// TIA Portal V16 export
// export: Created 2021-11-12T13:31:14.2602754Z, ExportSetting WithDefaults, DisplayName Totally Integrated Automation Portal, DisplayVersion V16 Update 3, DisplayName TIA Portal Version Control Interface, DisplayVersion V16 Update 2, DisplayName TIA Portal Openness, DisplayVersion V16 Update 3, DisplayName SINAMICS Startdrive Advanced, DisplayVersion V16 Update 5, DisplayName SINAMICS Startdrive G130, G150, S120, S150, SINAMICS MV, S210, DisplayVersion V16 Update 5, DisplayName SINAMICS Startdrive G110M, G120, G120C, G120D, G120P, G115D, DisplayVersion V16 Update 5, DisplayName STEP 7 Professional, DisplayVersion V16 Update 3, DisplayName STEP 7 Safety, DisplayVersion V16, DisplayName WinCC UA Professional, DisplayVersion V16 Update 3
FUNCTION_BLOCK "STD_EuchnerSafetySwitch2MBM"   // FB84, LAD
TITLE = Euchner safety switch 2 Main module / Euchner bezpečnostní zámek 2 hlavní modul
{ S7_Optimized_Access := 'TRUE' }
VERSION : 0.1
// MICE STD Function Block
// STD_EuchnerSafetySwitch2 MBM module
// 
// Version                             Creation date                       Created by
// 0.1                                     16.8.2019                                ZS
// stored: AutoNumber true, IsIECCheckEnabled false, IsRetainMemResEnabled false, MemoryReserve 100, SetENOAutomatically false, UDAEnableTagReadback false
   VAR_INPUT
      IS_ZoneM { ExternalAccessible := 'False'; ExternalVisible := 'False'; ExternalWritable := 'False'} : "UDT_Status_main";   // Main structure from zone / Main struktura ze zóny
      IS_ZoneS { ExternalAccessible := 'False'; ExternalVisible := 'False'; ExternalWritable := 'False'} : "UDT_Zone_Status_specific";   // Specific structure from zone / Specific struktura zóny
      IB1ResetLock : Bool;   // Reset errors and lock / Reset chyby a zamknutí
      IB1AlarmSuppress : Bool;   // Alarm suppression - external / Potlačení poruch
      IB_DoorMBMData : "UDT_MBM_Extended.Input";   // Vstupní data z modulu MBM / Input data from module
   END_VAR
   VAR_OUTPUT
      OS_Status : Struct
         Main : "UDT_Status_main";
         Specific : "UDT_EuchnerSafetySwitch2MBM_Status_Specific";
         Error : "UDT_Error01";
      END_STRUCT;
      OB_DoorMBMReset : Bool;   // Reset output byte for MBM module / Reset výstupního bitu pro MBM modul
   END_VAR
   VAR
      SS_Alarm : Struct   // Device alarms / Zařízení poruchy
         DoorMainModule : Bool;   // Door main module / Dveře hlavní modul
         DoorModule1 : Bool;   // Door module 1 / Dveře modul 1
         DoorModule2 : Bool;   // Dveře modul 2 / Door module 2
         DoorOverallSystem : Bool;   // Dveře nadřazený systém / Door overall system
         Res_0_4 : Bool;
         Res_0_5 : Bool;
         Res_0_6 : Bool;
         Res_0_7 : Bool;
         Res_1_0 : Bool;
         Res_1_1 : Bool;
         Res_1_2 : Bool;
         Res_1_3 : Bool;
         Res_1_4 : Bool;
         Res_1_5 : Bool;
         Res_1_6 : Bool;
         Res_1_7 : Bool;
      END_STRUCT;
      SS_Warning : Struct   // Device warnings / Zařízení varování
         Res_0_0 : Bool;
         Res_0_1 : Bool;
         Res_0_2 : Bool;
         Res_0_3 : Bool;
         Res_0_4 : Bool;
         Res_0_5 : Bool;
         Res_0_6 : Bool;
         Res_0_7 : Bool;
         Res_1_0 : Bool;
         Res_1_1 : Bool;
         Res_1_2 : Bool;
         Res_1_3 : Bool;
         Res_1_4 : Bool;
         Res_1_5 : Bool;
         Res_1_6 : Bool;
         Res_1_7 : Bool;
      END_STRUCT;
      SB1CollError : Bool;   // Collective error from device / Sumace poruchy zařízení
      ST_TONExtensAck { S7_SetPoint := 'True'} : TON_TIME;   // Časovač pro prodloužení pulsu / Timer for extension pulse
      SB_DoorMBMReset : Bool;   // Reset output byte for MBM module / Reset výstupního bitu pro MBM modulu
      SB1Reset : Bool;   // Reset errors and lock / Reset chyby a zamknutí
      SB1ResetEdge : Bool;   // Edge reset errors and lock / Hrana resetu poruchy a zamknutí
   END_VAR
   VAR_TEMP
      TS_Status : Struct
         Main : "UDT_Status_main";
         Specific : "UDT_EuchnerSafetySwitch2MBM_Status_Specific";
         Error : "UDT_Error01";
      END_STRUCT;
      TS_Command : "UDT_EuchnerSafetySwitch2MBM_Command";
      TS_Parameter : "UDT_EuchnerSafetySwitch2MBM_Parameter";
   END_VAR
   VAR_TEMP   // added for the SCL form of the ladder/FBD networks
      _w1 : Bool;
   END_VAR
BEGIN

REGION Network 1: Clear temporary TS_Status - Main, Specific / Mazání dočasných TS_Status - Main, Specific
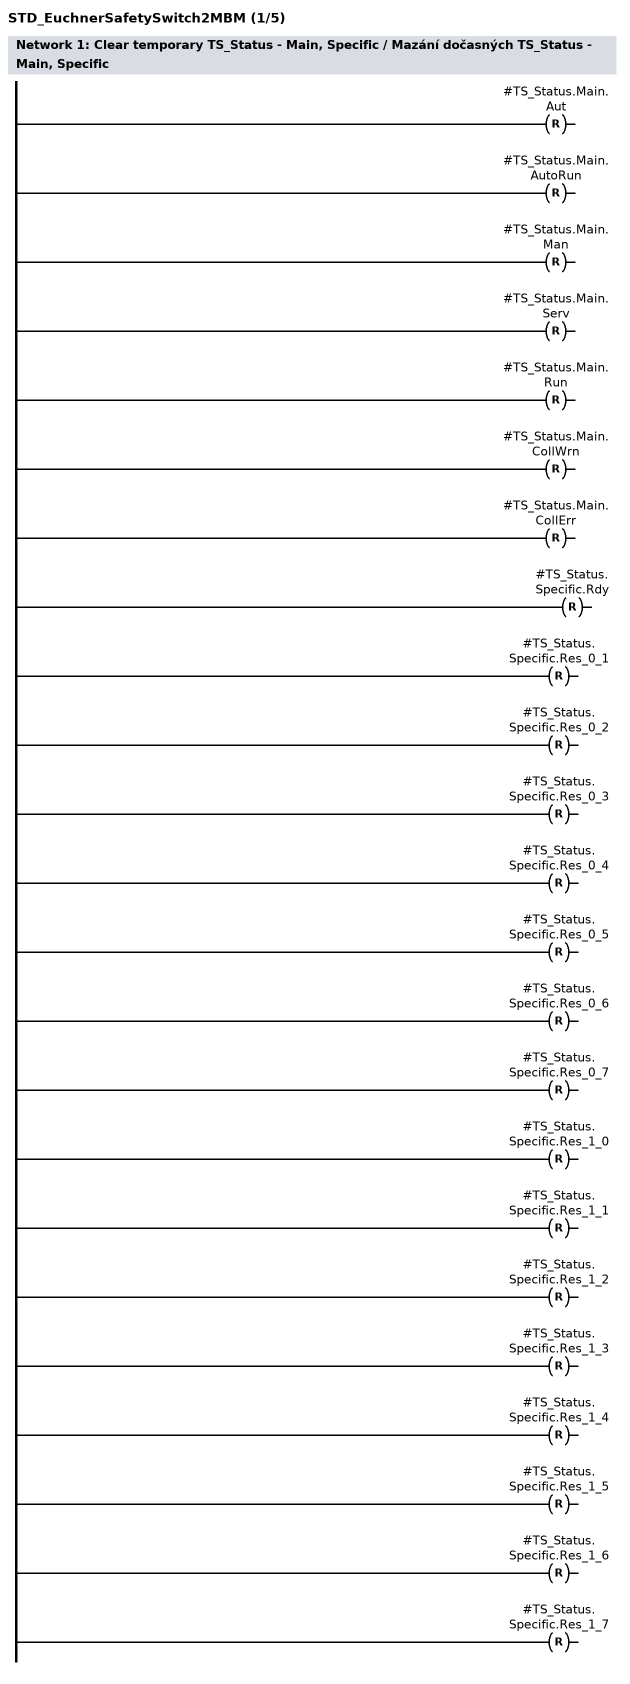
   RUNG wire#powerrail
      R_Coil( #TS_Status.Main.Aut )
   END_RUNG
   RUNG wire#powerrail
      R_Coil( #TS_Status.Main.AutoRun )
   END_RUNG
   RUNG wire#powerrail
      R_Coil( #TS_Status.Main.Man )
   END_RUNG
   RUNG wire#powerrail
      R_Coil( #TS_Status.Main.Serv )
   END_RUNG
   RUNG wire#powerrail
      R_Coil( #TS_Status.Main.Run )
   END_RUNG
   RUNG wire#powerrail
      R_Coil( #TS_Status.Main.CollWrn )
   END_RUNG
   RUNG wire#powerrail
      R_Coil( #TS_Status.Main.CollErr )
   END_RUNG
   RUNG wire#powerrail
      R_Coil( #TS_Status.Specific.Rdy )
   END_RUNG
   RUNG wire#powerrail
      R_Coil( #TS_Status.Specific.Res_0_1 )
   END_RUNG
   RUNG wire#powerrail
      R_Coil( #TS_Status.Specific.Res_0_2 )
   END_RUNG
   RUNG wire#powerrail
      R_Coil( #TS_Status.Specific.Res_0_3 )
   END_RUNG
   RUNG wire#powerrail
      R_Coil( #TS_Status.Specific.Res_0_4 )
   END_RUNG
   RUNG wire#powerrail
      R_Coil( #TS_Status.Specific.Res_0_5 )
   END_RUNG
   RUNG wire#powerrail
      R_Coil( #TS_Status.Specific.Res_0_6 )
   END_RUNG
   RUNG wire#powerrail
      R_Coil( #TS_Status.Specific.Res_0_7 )
   END_RUNG
   RUNG wire#powerrail
      R_Coil( #TS_Status.Specific.Res_1_0 )
   END_RUNG
   RUNG wire#powerrail
      R_Coil( #TS_Status.Specific.Res_1_1 )
   END_RUNG
   RUNG wire#powerrail
      R_Coil( #TS_Status.Specific.Res_1_2 )
   END_RUNG
   RUNG wire#powerrail
      R_Coil( #TS_Status.Specific.Res_1_3 )
   END_RUNG
   RUNG wire#powerrail
      R_Coil( #TS_Status.Specific.Res_1_4 )
   END_RUNG
   RUNG wire#powerrail
      R_Coil( #TS_Status.Specific.Res_1_5 )
   END_RUNG
   RUNG wire#powerrail
      R_Coil( #TS_Status.Specific.Res_1_6 )
   END_RUNG
   RUNG wire#powerrail
      R_Coil( #TS_Status.Specific.Res_1_7 )
   END_RUNG
   // the same network as SCL:
   #TS_Status.Main.Aut := FALSE;
   #TS_Status.Main.AutoRun := FALSE;
   #TS_Status.Main.Man := FALSE;
   #TS_Status.Main.Serv := FALSE;
   #TS_Status.Main.Run := FALSE;
   #TS_Status.Main.CollWrn := FALSE;
   #TS_Status.Main.CollErr := FALSE;
   #TS_Status.Specific.Rdy := FALSE;
   #TS_Status.Specific.Res_0_1 := FALSE;
   #TS_Status.Specific.Res_0_2 := FALSE;
   #TS_Status.Specific.Res_0_3 := FALSE;
   #TS_Status.Specific.Res_0_4 := FALSE;
   #TS_Status.Specific.Res_0_5 := FALSE;
   #TS_Status.Specific.Res_0_6 := FALSE;
   #TS_Status.Specific.Res_0_7 := FALSE;
   #TS_Status.Specific.Res_1_0 := FALSE;
   #TS_Status.Specific.Res_1_1 := FALSE;
   #TS_Status.Specific.Res_1_2 := FALSE;
   #TS_Status.Specific.Res_1_3 := FALSE;
   #TS_Status.Specific.Res_1_4 := FALSE;
   #TS_Status.Specific.Res_1_5 := FALSE;
   #TS_Status.Specific.Res_1_6 := FALSE;
   #TS_Status.Specific.Res_1_7 := FALSE;
END_REGION

REGION Network 2: Door Ack / Dveře potvrzení
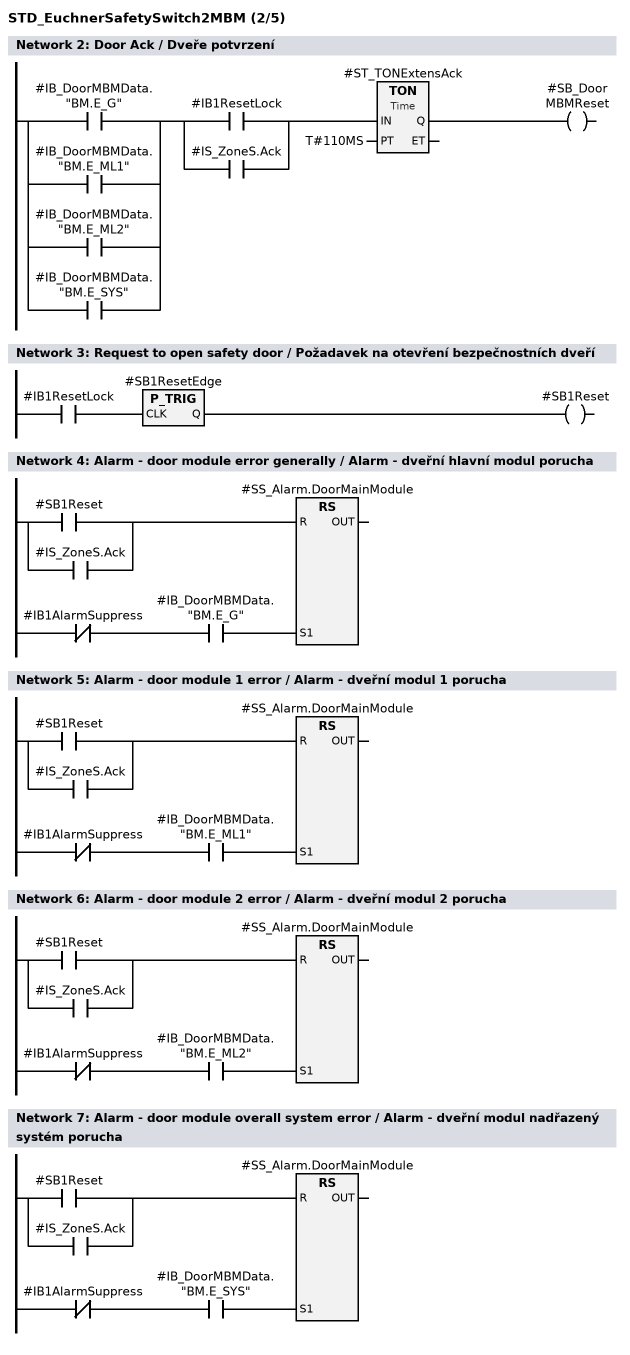
   RUNG wire#powerrail
      Contact( #IB_DoorMBMData."BM.E_G" )
      wire#w1
      Contact( #IB1ResetLock )
      wire#w2
      { S7_Templates := "time_type := Time" } #ST_TONExtensAck.TON(pt := T#110MS, et =>)
      Coil( #SB_DoorMBMReset )
   END_RUNG
   RUNG wire#powerrail
      Contact( #IB_DoorMBMData."BM.E_ML1" )
   END_RUNG wire#w1
   RUNG wire#powerrail
      Contact( #IB_DoorMBMData."BM.E_ML2" )
   END_RUNG wire#w1
   RUNG wire#powerrail
      Contact( #IB_DoorMBMData."BM.E_SYS" )
   END_RUNG wire#w1
   RUNG wire#w1
      Contact( #IS_ZoneS.Ack )
   END_RUNG wire#w2
   // the same network as SCL:
   #ST_TONExtensAck(IN := (#IB_DoorMBMData."BM.E_G" OR #IB_DoorMBMData."BM.E_ML1" OR #IB_DoorMBMData."BM.E_ML2" OR #IB_DoorMBMData."BM.E_SYS") AND (#IB1ResetLock OR #IS_ZoneS.Ack),   // TON
                    PT := T#110MS);
   #SB_DoorMBMReset := #ST_TONExtensAck.Q;
END_REGION

REGION Network 3: Request to open safety door / Požadavek na otevření bezpečnostních dveří
   RUNG wire#powerrail
      Contact( #IB1ResetLock )
      P_Trig( #SB1ResetEdge )
      Coil( #SB1Reset )
   END_RUNG
   // the same network as SCL:
   #_w1 := #IB1ResetLock AND NOT #SB1ResetEdge;   // rising edge
   #SB1ResetEdge := #IB1ResetLock;
   #SB1Reset := #_w1;
END_REGION

REGION Network 4: Alarm - door module error generally / Alarm - dveřní hlavní modul porucha
   RUNG wire#powerrail
      Contact( #SB1Reset )
      wire#w1
      S_RS(operand := #SS_Alarm.DoorMainModule, s1 := wire#w2)
   END_RUNG
   RUNG wire#powerrail
      Contact( #IS_ZoneS.Ack )
   END_RUNG wire#w1
   RUNG wire#powerrail
      I_Contact( #IB1AlarmSuppress )
      Contact( #IB_DoorMBMData."BM.E_G" )
   END_RUNG wire#w2
   // the same network as SCL:
   IF #SB1Reset OR #IS_ZoneS.Ack THEN
       #SS_Alarm.DoorMainModule := FALSE;   // RS flip-flop
   END_IF;
   IF NOT #IB1AlarmSuppress AND #IB_DoorMBMData."BM.E_G" THEN #SS_Alarm.DoorMainModule := TRUE; END_IF;
END_REGION

REGION Network 5: Alarm - door module 1 error / Alarm - dveřní modul 1 porucha
   RUNG wire#powerrail
      Contact( #SB1Reset )
      wire#w1
      S_RS(operand := #SS_Alarm.DoorMainModule, s1 := wire#w2)
   END_RUNG
   RUNG wire#powerrail
      Contact( #IS_ZoneS.Ack )
   END_RUNG wire#w1
   RUNG wire#powerrail
      I_Contact( #IB1AlarmSuppress )
      Contact( #IB_DoorMBMData."BM.E_ML1" )
   END_RUNG wire#w2
   // the same network as SCL:
   IF #SB1Reset OR #IS_ZoneS.Ack THEN
       #SS_Alarm.DoorMainModule := FALSE;   // RS flip-flop
   END_IF;
   IF NOT #IB1AlarmSuppress AND #IB_DoorMBMData."BM.E_ML1" THEN #SS_Alarm.DoorMainModule := TRUE; END_IF;
END_REGION

REGION Network 6: Alarm - door module 2 error / Alarm - dveřní modul 2 porucha
   RUNG wire#powerrail
      Contact( #SB1Reset )
      wire#w1
      S_RS(operand := #SS_Alarm.DoorMainModule, s1 := wire#w2)
   END_RUNG
   RUNG wire#powerrail
      Contact( #IS_ZoneS.Ack )
   END_RUNG wire#w1
   RUNG wire#powerrail
      I_Contact( #IB1AlarmSuppress )
      Contact( #IB_DoorMBMData."BM.E_ML2" )
   END_RUNG wire#w2
   // the same network as SCL:
   IF #SB1Reset OR #IS_ZoneS.Ack THEN
       #SS_Alarm.DoorMainModule := FALSE;   // RS flip-flop
   END_IF;
   IF NOT #IB1AlarmSuppress AND #IB_DoorMBMData."BM.E_ML2" THEN #SS_Alarm.DoorMainModule := TRUE; END_IF;
END_REGION

REGION Network 7: Alarm - door module overall system error / Alarm - dveřní modul nadřazený systém porucha
   RUNG wire#powerrail
      Contact( #SB1Reset )
      wire#w1
      S_RS(operand := #SS_Alarm.DoorMainModule, s1 := wire#w2)
   END_RUNG
   RUNG wire#powerrail
      Contact( #IS_ZoneS.Ack )
   END_RUNG wire#w1
   RUNG wire#powerrail
      I_Contact( #IB1AlarmSuppress )
      Contact( #IB_DoorMBMData."BM.E_SYS" )
   END_RUNG wire#w2
   // the same network as SCL:
   IF #SB1Reset OR #IS_ZoneS.Ack THEN
       #SS_Alarm.DoorMainModule := FALSE;   // RS flip-flop
   END_IF;
   IF NOT #IB1AlarmSuppress AND #IB_DoorMBMData."BM.E_SYS" THEN #SS_Alarm.DoorMainModule := TRUE; END_IF;
END_REGION

REGION Network 8: Collective error of device / Sumace poruchy zařízení
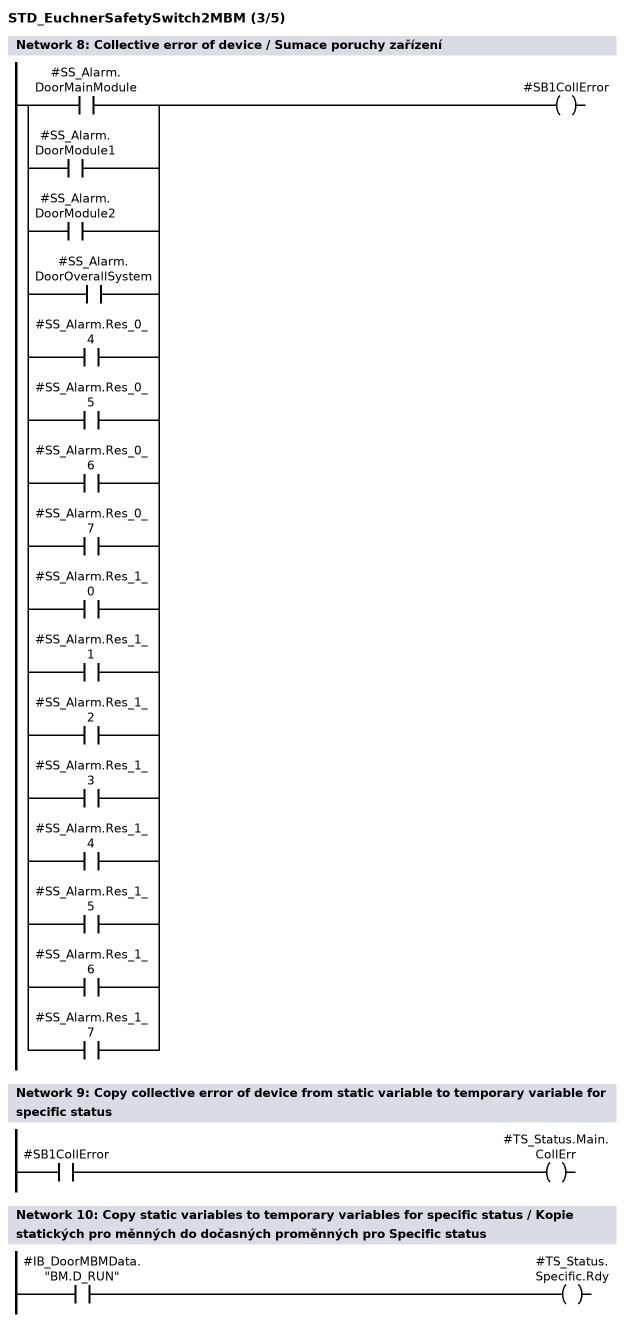
   RUNG wire#powerrail
      Contact( #SS_Alarm.DoorMainModule )
      wire#w1
      Coil( #SB1CollError )
   END_RUNG
   RUNG wire#powerrail
      Contact( #SS_Alarm.DoorModule1 )
   END_RUNG wire#w1
   RUNG wire#powerrail
      Contact( #SS_Alarm.DoorModule2 )
   END_RUNG wire#w1
   RUNG wire#powerrail
      Contact( #SS_Alarm.DoorOverallSystem )
   END_RUNG wire#w1
   RUNG wire#powerrail
      Contact( #SS_Alarm.Res_0_4 )
   END_RUNG wire#w1
   RUNG wire#powerrail
      Contact( #SS_Alarm.Res_0_5 )
   END_RUNG wire#w1
   RUNG wire#powerrail
      Contact( #SS_Alarm.Res_0_6 )
   END_RUNG wire#w1
   RUNG wire#powerrail
      Contact( #SS_Alarm.Res_0_7 )
   END_RUNG wire#w1
   RUNG wire#powerrail
      Contact( #SS_Alarm.Res_1_0 )
   END_RUNG wire#w1
   RUNG wire#powerrail
      Contact( #SS_Alarm.Res_1_1 )
   END_RUNG wire#w1
   RUNG wire#powerrail
      Contact( #SS_Alarm.Res_1_2 )
   END_RUNG wire#w1
   RUNG wire#powerrail
      Contact( #SS_Alarm.Res_1_3 )
   END_RUNG wire#w1
   RUNG wire#powerrail
      Contact( #SS_Alarm.Res_1_4 )
   END_RUNG wire#w1
   RUNG wire#powerrail
      Contact( #SS_Alarm.Res_1_5 )
   END_RUNG wire#w1
   RUNG wire#powerrail
      Contact( #SS_Alarm.Res_1_6 )
   END_RUNG wire#w1
   RUNG wire#powerrail
      Contact( #SS_Alarm.Res_1_7 )
   END_RUNG wire#w1
   // the same network as SCL:
   #SB1CollError := #SS_Alarm.DoorMainModule OR #SS_Alarm.DoorModule1 OR #SS_Alarm.DoorModule2 OR #SS_Alarm.DoorOverallSystem OR #SS_Alarm.Res_0_4 OR #SS_Alarm.Res_0_5 OR #SS_Alarm.Res_0_6 OR #SS_Alarm.Res_0_7 OR #SS_Alarm.Res_1_0 OR #SS_Alarm.Res_1_1 OR #SS_Alarm.Res_1_2 OR #SS_Alarm.Res_1_3 OR #SS_Alarm.Res_1_4 OR #SS_Alarm.Res_1_5 OR #SS_Alarm.Res_1_6 OR #SS_Alarm.Res_1_7;
END_REGION

REGION Network 9: Copy collective error of device from static variable to temporary variable for specific status
   RUNG wire#powerrail
      Contact( #SB1CollError )
      Coil( #TS_Status.Main.CollErr )
   END_RUNG
   // the same network as SCL:
   #TS_Status.Main.CollErr := #SB1CollError;
END_REGION

REGION Network 10: Copy static variables to temporary variables for specific status / Kopie statických pro měnných do dočasných proměnných pro Specific status
   RUNG wire#powerrail
      Contact( #IB_DoorMBMData."BM.D_RUN" )
      Coil( #TS_Status.Specific.Rdy )
   END_RUNG
   // the same network as SCL:
   #TS_Status.Specific.Rdy := #IB_DoorMBMData."BM.D_RUN";
END_REGION

REGION Network 11: Alarms - copy to output structure / Porucha - kopie do výstupní struktury
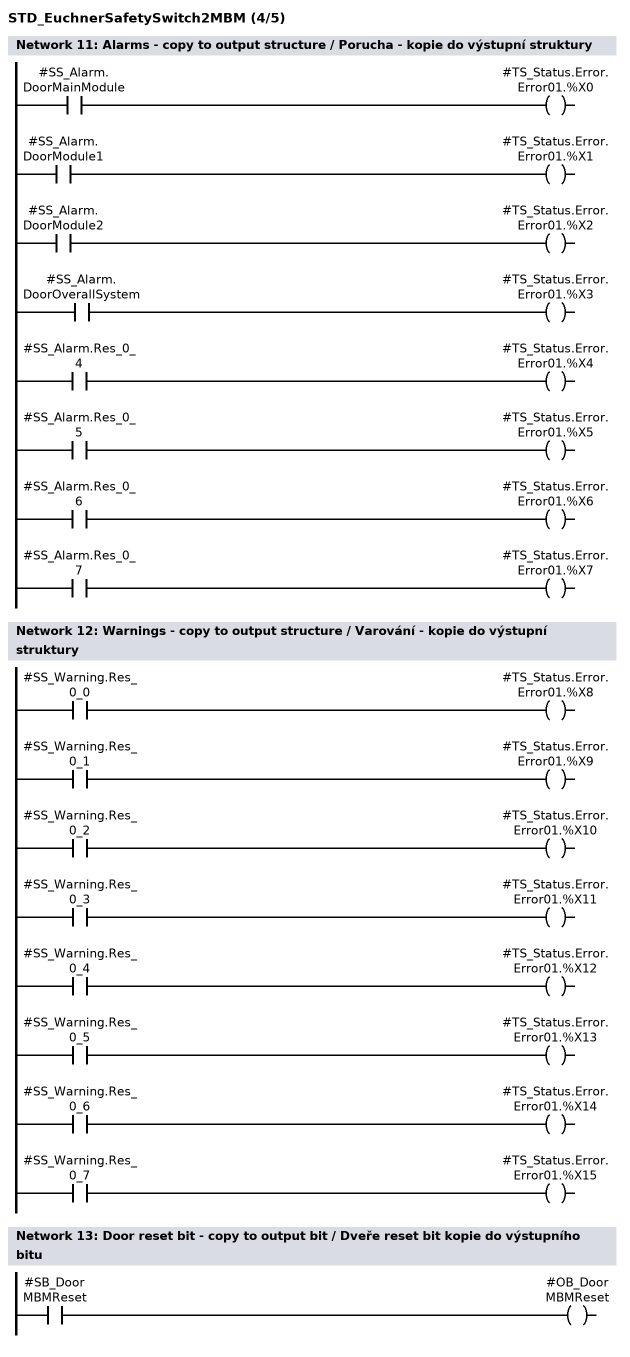
   RUNG wire#powerrail
      Contact( #SS_Alarm.DoorMainModule )
      Coil( #TS_Status.Error.Error01.%X0 )
   END_RUNG
   RUNG wire#powerrail
      Contact( #SS_Alarm.DoorModule1 )
      Coil( #TS_Status.Error.Error01.%X1 )
   END_RUNG
   RUNG wire#powerrail
      Contact( #SS_Alarm.DoorModule2 )
      Coil( #TS_Status.Error.Error01.%X2 )
   END_RUNG
   RUNG wire#powerrail
      Contact( #SS_Alarm.DoorOverallSystem )
      Coil( #TS_Status.Error.Error01.%X3 )
   END_RUNG
   RUNG wire#powerrail
      Contact( #SS_Alarm.Res_0_4 )
      Coil( #TS_Status.Error.Error01.%X4 )
   END_RUNG
   RUNG wire#powerrail
      Contact( #SS_Alarm.Res_0_5 )
      Coil( #TS_Status.Error.Error01.%X5 )
   END_RUNG
   RUNG wire#powerrail
      Contact( #SS_Alarm.Res_0_6 )
      Coil( #TS_Status.Error.Error01.%X6 )
   END_RUNG
   RUNG wire#powerrail
      Contact( #SS_Alarm.Res_0_7 )
      Coil( #TS_Status.Error.Error01.%X7 )
   END_RUNG
   // the same network as SCL:
   #TS_Status.Error.Error01.%X0 := #SS_Alarm.DoorMainModule;
   #TS_Status.Error.Error01.%X1 := #SS_Alarm.DoorModule1;
   #TS_Status.Error.Error01.%X2 := #SS_Alarm.DoorModule2;
   #TS_Status.Error.Error01.%X3 := #SS_Alarm.DoorOverallSystem;
   #TS_Status.Error.Error01.%X4 := #SS_Alarm.Res_0_4;
   #TS_Status.Error.Error01.%X5 := #SS_Alarm.Res_0_5;
   #TS_Status.Error.Error01.%X6 := #SS_Alarm.Res_0_6;
   #TS_Status.Error.Error01.%X7 := #SS_Alarm.Res_0_7;
END_REGION

REGION Network 12: Warnings - copy to output structure / Varování - kopie do výstupní struktury
   RUNG wire#powerrail
      Contact( #SS_Warning.Res_0_0 )
      Coil( #TS_Status.Error.Error01.%X8 )
   END_RUNG
   RUNG wire#powerrail
      Contact( #SS_Warning.Res_0_1 )
      Coil( #TS_Status.Error.Error01.%X9 )
   END_RUNG
   RUNG wire#powerrail
      Contact( #SS_Warning.Res_0_2 )
      Coil( #TS_Status.Error.Error01.%X10 )
   END_RUNG
   RUNG wire#powerrail
      Contact( #SS_Warning.Res_0_3 )
      Coil( #TS_Status.Error.Error01.%X11 )
   END_RUNG
   RUNG wire#powerrail
      Contact( #SS_Warning.Res_0_4 )
      Coil( #TS_Status.Error.Error01.%X12 )
   END_RUNG
   RUNG wire#powerrail
      Contact( #SS_Warning.Res_0_5 )
      Coil( #TS_Status.Error.Error01.%X13 )
   END_RUNG
   RUNG wire#powerrail
      Contact( #SS_Warning.Res_0_6 )
      Coil( #TS_Status.Error.Error01.%X14 )
   END_RUNG
   RUNG wire#powerrail
      Contact( #SS_Warning.Res_0_7 )
      Coil( #TS_Status.Error.Error01.%X15 )
   END_RUNG
   // the same network as SCL:
   #TS_Status.Error.Error01.%X8 := #SS_Warning.Res_0_0;
   #TS_Status.Error.Error01.%X9 := #SS_Warning.Res_0_1;
   #TS_Status.Error.Error01.%X10 := #SS_Warning.Res_0_2;
   #TS_Status.Error.Error01.%X11 := #SS_Warning.Res_0_3;
   #TS_Status.Error.Error01.%X12 := #SS_Warning.Res_0_4;
   #TS_Status.Error.Error01.%X13 := #SS_Warning.Res_0_5;
   #TS_Status.Error.Error01.%X14 := #SS_Warning.Res_0_6;
   #TS_Status.Error.Error01.%X15 := #SS_Warning.Res_0_7;
END_REGION

REGION Network 13: Door reset bit - copy to output bit / Dveře reset bit kopie do výstupního bitu
   RUNG wire#powerrail
      Contact( #SB_DoorMBMReset )
      Coil( #OB_DoorMBMReset )
   END_RUNG
   // the same network as SCL:
   #OB_DoorMBMReset := #SB_DoorMBMReset;
END_REGION

REGION Network 14: Copy temporary variables to output variables / Kopie dočasných proměnných do výstupních proměnných
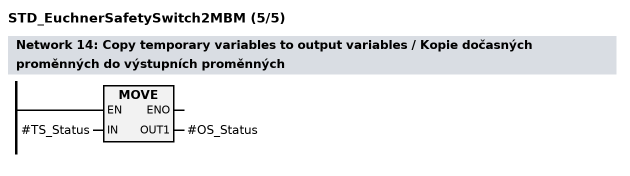
   RUNG wire#powerrail
      Move(in := #TS_Status, out1 => #OS_Status)
   END_RUNG
   // the same network as SCL:
   #OS_Status := #TS_Status;
END_REGION
END_FUNCTION_BLOCK
